// TIA Portal V19 export
DATA_BLOCK "Area01_Messages"   // DB55
// stored: MemoryReserve 100
   VAR
      "A" : Struct
         Msg : Array[1..352] of Bool;
         Hmi : Array[1..22] of Word;
         Ack : Array[1..22] of Word;
      END_STRUCT;
      W : Struct
         Msg : Array[1..384] of Bool;
         Hmi : Array[1..24] of Word;
         Ack : Array[1..24] of Word;
      END_STRUCT;
   END_VAR
BEGIN
   // "A".Msg[2] : h
   // "A".Msg[3] : hsfdd
END_DATA_BLOCK
